{attribute 'GeneratedUsingTerminal: EL4712--0000'}
{attribute addProperty BoxType "EL4712--0000"}
{attribute addProperty Id "Ch2_ValueAT %Q*INT2"}
{attribute addProperty CRC "4033423121"}
{attribute addProperty Size "2"}
TYPE Ch2_Sample_F0692711 :
STRUCT
	{attribute addProperty Name "Ch2_Value"}
	Ch2_Value AT %Q* : INT;
END_STRUCT
END_TYPE

(* stored: Version 1.2.0.0, ProductVersion 3.1.4024.9
   DUT Ch2_Sample_F0692711: Id {c4169dc0-0840-4fe5-a1a3-47d65b7f6830} *)
